FUNCTION_BLOCK HeartBeat_HMI (* Service Interface Function Block Type *)
  (* Standard: 61499-2 *)
  (* Version 0.0, 25/02/2022, SESA197029, template *)
  PACKAGE SE.Nereda;
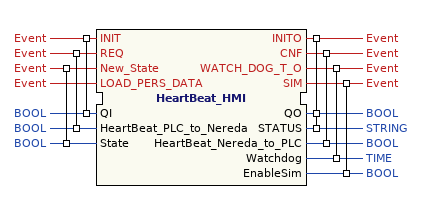
  EVENT_INPUT
    INIT WITH QI;
    REQ WITH HeartBeat_PLC_to_Nereda;
    New_State WITH State;
    LOAD_PERS_DATA;
  END_EVENT
  EVENT_OUTPUT
    INITO WITH QO, STATUS;
    CNF WITH HeartBeat_Nereda_to_PLC;
    WATCH_DOG_T_O WITH Watchdog;
    SIM WITH EnableSim;
  END_EVENT
  VAR_INPUT
    QI : BOOL;
    HeartBeat_PLC_to_Nereda : BOOL;
    State : BOOL;
  END_VAR
  VAR_OUTPUT
    QO : BOOL; (* Event Output Qualifier *)
    STATUS : STRING; (* Service Status *)
    HeartBeat_Nereda_to_PLC : BOOL;
    Watchdog : TIME;
    EnableSim : BOOL;
  END_VAR
  SERVICE /
    SEQUENCE 
    END_SEQUENCE
  END_SERVICE
END_FUNCTION_BLOCK
